{attribute 'qualified_only'}
{attribute 'strict'}
TYPE PLCopenCallState :
(
	PLCOPEN_FUB_IDLE := 0,
	PLCOPEN_FUB_NEW_COMMAND,
	PLCOPEN_FUB_ABORTED,
	PLCOPEN_FUB_ABORT_OLD,
	PLCOPEN_FUB_STATUS,
	PLCOPEN_FUB_WRITE_PAR,
	PLCOPEN_FUB_SET_COMMAND,
	PLCOPEN_FUB_WORKING,
	PLCOPEN_FUB_CLEANUP,
	PLCOPEN_FUB_DONE
);
END_TYPE

(* stored: Version 1.1.0.1
   EnumerationTextList PLCopenCallState: Id {3ae6e054-32d2-4fc8-9116-cc770a82905a} *)
